FUNCTION_BLOCK _STRING_TestSuite EXTENDS TcUnit.FB_TestSuite
VAR
END_VAR

TestAddress();
TestClearReference();
TestClone();
TestIecTypeReturnsExpected();
TestMakeReferenceToFollowsReference();
TestMakeReferenceToUpdatesReference();
TestSize();
TestValueReturnsExpectedAfterInit();
TestValueReturnsExpectedAfterChange();
TestSerializeTypeWith();
TestSerializeWith();
TestTryDeserializeFrom();
TestTryMakeReferenceToFollowsReference();
TestTryMakeReferenceToUpdatesReference();

METHOD PUBLIC TestAddress
VAR
    _type : _STRING('');
    notExpected : PVOID := 0;
    actual : PVOID;
END_VAR
TEST('TestAddress');

actual := _type.Address;

AssertFalse(
    Condition := (notExpected = actual),
    Message := 'Type did not return a valid address.'
);

TEST_FINISHED();
END_METHOD

METHOD PUBLIC TestClearReference
VAR
    _type : _STRING('');
	target : T_MaxString := '';
    expected : T_MaxString := '';
    actual : T_MaxString;
END_VAR
TEST('TestClearReference');

_type.MakeReferenceTo(target);
_type.ClearReference();
target := '123';

actual := _type.Value;

AssertEquals_STRING(
    Expected := expected,
    Actual := actual,
    Message := 'Value did not follow target change'
);

TEST_FINISHED();
END_METHOD

METHOD PUBLIC TestClone
VAR
    _type : _STRING('123');
	clone : I_Datatype;
	isValidClone : BOOL;
	compareResult : DINT;
END_VAR
TEST('TestClone');

clone := _type.Clone();

isValidClone := clone <> 0;

IF isValidClone THEN
	compareResult := memcmp(_type.Address, clone.Address, clone.Size);
END_IF

AssertTrue(
	Condition := isValidClone,
	Message := 'Clone did not produce a clone'
);

AssertEquals_DINT(
	Expected := 0,
    Actual := compareResult,
    Message := 'Clone did not return a valid clone.'
);

clone.Dispose();

TEST_FINISHED();
END_METHOD

METHOD PUBLIC TestIecTypeReturnsExpected
VAR
    _type : _STRING('');
    expected : STRING := 'STRING';
    actual : STRING;
END_VAR
TEST('TestIecTypeReturnsExpected');

actual := _type.Datatype;

AssertEquals_STRING(
    Expected := expected,
    Actual := actual,
    Message := 'Type did not return correct iec type.'
);

TEST_FINISHED();
END_METHOD

METHOD PUBLIC TestMakeReferenceToFollowsReference
VAR
    _type : _STRING('');
	target : T_MaxString := '';
    expected : T_MaxString := '123';
    actual : T_MaxString;
END_VAR
TEST('TestMakeReferenceToFollowsReference');

_type.MakeReferenceTo(target);
target := '123';

actual := _type.Value;

AssertEquals_STRING(
    Expected := expected,
    Actual := actual,
    Message := 'Value did not follow target change'
);

TEST_FINISHED();
END_METHOD

METHOD PUBLIC TestMakeReferenceToUpdatesReference
VAR
    _type : _STRING('');
	target : T_MaxString := '';
    expected : T_MaxString := '123';
    actual : T_MaxString;
END_VAR
TEST('TestMakeReferenceToUpdatesReference');

_type.MakeReferenceTo(target);
_type.Value := '123';

actual := target;

AssertEquals_STRING(
    Expected := expected,
    Actual := actual,
    Message := 'Value did not update target'
);

TEST_FINISHED();
END_METHOD

METHOD PUBLIC TestSerializeTypeWith
VAR
    _type : _STRING('');
    serializer : JsonSerializer;
    expected : STRING := '{"datatype":"STRING"}';
    actual : STRING(500);
END_VAR
TEST('TestSerializeTypeWith');

serializer.Reset();
_type.SerializeTypeWith(serializer);
serializer.TryGetSerializedData(ADR(actual), SIZEOF(actual));

AssertEquals_STRING(
    Expected := expected,
    Actual := actual,
    Message := 'Serialization of type did not return correct string.'
);

TEST_FINISHED();
END_METHOD

METHOD PUBLIC TestSerializeWith
VAR
    _type : _STRING('abcdefghijklmnopqrstuvwxyzABCDEFGHIJKLMNOPQRSTUVWXYZ01234567890');
    serializer : JsonSerializer;
    expected : STRING := '"abcdefghijklmnopqrstuvwxyzABCDEFGHIJKLMNOPQRSTUVWXYZ01234567890"';
    actual : STRING(500);
END_VAR
TEST('TestSerializeWith');

serializer.Reset();
_type.SerializeWith(serializer);
serializer.TryGetSerializedData(ADR(actual), SIZEOF(actual));

AssertEquals_STRING(
    Expected := expected,
    Actual := actual,
    Message := 'Serialization of type data did not return correct string.'
);

TEST_FINISHED();
END_METHOD

METHOD PUBLIC TestSize
VAR
    _type : _STRING('');
    expected : UDINT := SIZEOF(T_MaxString);
    actual : UDINT;
END_VAR
TEST('TestSize');

actual := _type.Size;

AssertEquals_UDINT(
    Expected := Expected,
    Actual := actual,
    Message := 'Type did not return the correct size.'
);

TEST_FINISHED();
END_METHOD

METHOD PUBLIC TestTryDeserializeFrom
VAR
    deserializer : JsonDeserializer;
    feedback : DeserializerFeedback;
    json : STRING := '"abcdefghijklmnopqrstuvwxyzABCDEFGHIJKLMNOPQRSTUVWXYZ01234567890"';
    _type : _STRING('');
    expected : T_MaxString := 'abcdefghijklmnopqrstuvwxyzABCDEFGHIJKLMNOPQRSTUVWXYZ01234567890';
    actual : T_MaxString;
 END_VAR
TEST('TestTryDeserializeFrom');

deserializer.Reset();
deserializer.TryLoad(json);
_type.TryDeserializeFrom(Deserializer, Feedback);

actual := _type.Value;

AssertEquals_STRING(
    Expected := expected,
    Actual := actual,
    Message := 'Type did not deserialize correctly.'
);

TEST_FINISHED();
END_METHOD

METHOD PUBLIC TestTryMakeReferenceToFollowsReference
VAR
    _type : _STRING('');
	target : _STRING('');
    expected : T_MaxString := '123';
    actual : T_MaxString;
END_VAR
TEST('TestTryMakeReferenceToFollowsReference');

_type.TryMakeReferenceTo(target);
target.Value := '123';

actual := _type.Value;

AssertEquals_STRING(
    Expected := expected,
    Actual := actual,
    Message := 'Value did not follow target change'
);

TEST_FINISHED();
END_METHOD

METHOD PUBLIC TestTryMakeReferenceToUpdatesReference
VAR
    _type : _STRING('');
	target : _STRING('');
    expected : T_MaxString := '123';
    actual : T_MaxString;
END_VAR
TEST('TestTryMakeReferenceToUpdatesReference');

_type.TryMakeReferenceTo(target);
_type.Value := '123';

actual := target.Value;

AssertEquals_STRING(
    Expected := expected,
    Actual := actual,
    Message := 'Value did not update target'
);

TEST_FINISHED();
END_METHOD

METHOD PUBLIC TestValueReturnsExpectedAfterChange
VAR
    _type : _STRING('');
    expected : T_MaxString := '123';
    actual : T_MaxString;
END_VAR
TEST('TestValueReturnsExpectedAfterChange');

_type.Value := '123';

actual := _type.Value;

AssertEquals_STRING(
    Expected := expected,
    Actual := actual,
    Message := 'Expected value not returned after change.'
);

TEST_FINISHED();
END_METHOD

METHOD PUBLIC TestValueReturnsExpectedAfterInit
VAR
    _type : _STRING('123');
    expected : T_MaxString := '123';
    actual : T_MaxString;
END_VAR
TEST('TestValueReturnsExpectedAfterInit');

actual := _type.Value;

AssertEquals_STRING(
    Expected := expected,
    Actual := actual,
    Message := 'Expected value not returned after Init.'
);

TEST_FINISHED();
END_METHOD

END_FUNCTION_BLOCK

(* stored: Version 1.1.0.1, ProductVersion 3.1.4024.12
   POU _STRING_TestSuite: Id {0b5fd00e-93dc-04d6-0518-ff531f9e7455}, SpecialFunc None
   Method TestAddress: Id {9d6ed495-e732-0ba5-2a3d-165e98a18aee}
   Method TestClearReference: Id {1af3c089-3411-04d4-3d8c-ba68a8a674d9}
   Method TestClone: Id {ed3d05de-6d7c-077b-37d4-dee196bece56}
   Method TestIecTypeReturnsExpected: Id {770f8363-3fb1-09ee-36e9-78fee07f030a}
   Method TestMakeReferenceToFollowsReference: Id {015ccb70-62c2-0f31-2aa1-fe22ba483b75}
   Method TestMakeReferenceToUpdatesReference: Id {cc9a830f-e0a7-0153-035c-dc83a60747f0}
   Method TestSerializeTypeWith: Id {6e5ffb7c-75a4-0d5c-1fde-78b371752859}
   Method TestSerializeWith: Id {b483d28a-1d85-021b-2a14-6bc9ba918f39}
   Method TestSize: Id {c03db28a-258e-01dc-377c-f42af4c430a0}
   Method TestTryDeserializeFrom: Id {b9c9105d-0d7b-0b9b-0fa9-91ad7e703bdc}
   Method TestTryMakeReferenceToFollowsReference: Id {60cdd5d4-5cd4-0360-1908-16223dd3dec6}
   Method TestTryMakeReferenceToUpdatesReference: Id {6df02952-d9b5-0a8c-26df-dbedfb9c32cf}
   Method TestValueReturnsExpectedAfterChange: Id {40ea4506-b078-0875-2fd3-b848745a9b2c}
   Method TestValueReturnsExpectedAfterInit: Id {28bc8ac9-34cb-0e35-040a-e05189f4be5c} *)
